// TIA Portal V15.1 export
// export: Created 2024-06-21T08:40:52.3398927Z, ExportSetting WithDefaults, DisplayName Totally Integrated Automation Portal, DisplayVersion V15.1 Update 5, DisplayName TIA Portal Openness, DisplayVersion V15.1 Update 5, DisplayName SINAMICS Startdrive Advanced, DisplayVersion V15.1, DisplayName G130, G150, S120, S150, SINAMICS MV, S210, DisplayVersion V15.1, DisplayName G110M, G120, G120C, G120D, G120P, DisplayVersion V15.1, DisplayName STEP 7 Professional, DisplayVersion V15.1 Update 5, DisplayName STEP 7 Safety, DisplayVersion V15.1, DisplayName WinCC Professional, DisplayVersion V15.1 Update 5, DisplayName SIMATIC Visualization Architect, DisplayVersion V15.1
FUNCTION "F209230ZS01Logic" : Void   // FC7031, F_FBD
TITLE = Safety Inputs ZMProc / Safety Logic 209230ZS01
{ S7_Optimized_Access := 'TRUE' }
VERSION : 0.1
// stored: AutoNumber false, IsIECCheckEnabled false, UDAEnableTagReadback false
   VAR_TEMP   // added for the SCL form of the ladder/FBD networks
      _w1 : Bool;
   END_VAR
BEGIN

REGION Network 1: **** 4.4 - Machine Status - Calculation **** Emergency Stop OK
   // Emergency Stop Ok When All Safety Inputs Are Ok
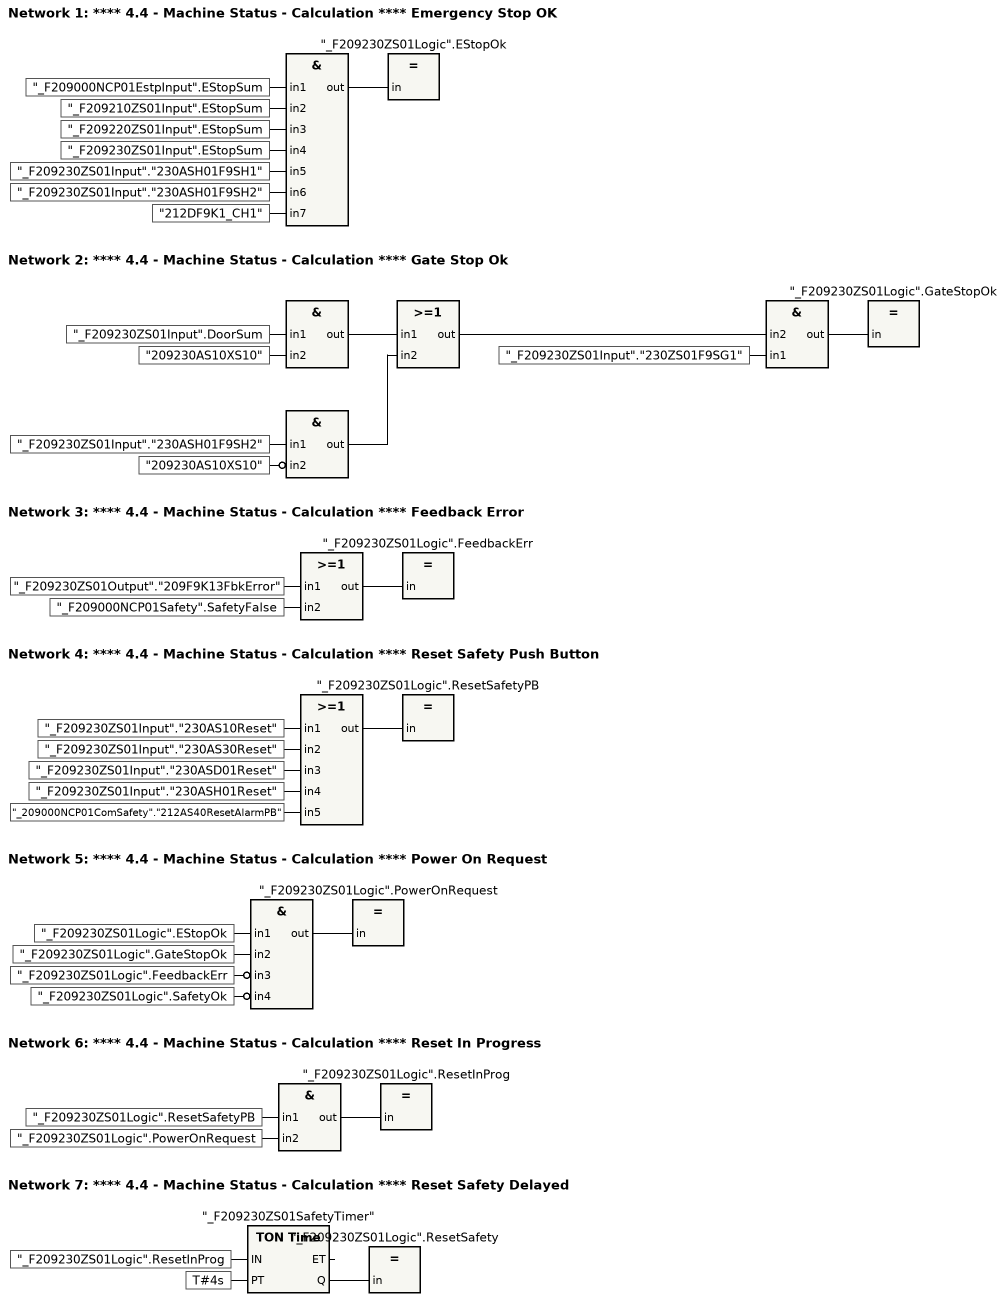
   "_F209230ZS01Logic".EStopOk := "_F209000NCP01EstpInput".EStopSum AND "_F209210ZS01Input".EStopSum AND "_F209220ZS01Input".EStopSum AND "_F209230ZS01Input".EStopSum AND "_F209230ZS01Input"."230ASH01F9SH1" AND "_F209230ZS01Input"."230ASH01F9SH2" AND "212DF9K1_CH1";
END_REGION

REGION Network 2: **** 4.4 - Machine Status - Calculation **** Gate Stop Ok
   // Gate Stop Ok
   "_F209230ZS01Logic".GateStopOk := (("_F209230ZS01Input".DoorSum AND "209230AS10XS10") OR ("_F209230ZS01Input"."230ASH01F9SH2" AND NOT "209230AS10XS10")) AND "_F209230ZS01Input"."230ZS01F9SG1";
END_REGION

REGION Network 3: **** 4.4 - Machine Status - Calculation **** Feedback Error
   // Feedback Error
   "_F209230ZS01Logic".FeedbackErr := "_F209230ZS01Output"."209F9K13FbkError" OR "_F209000NCP01Safety".SafetyFalse;
END_REGION

REGION Network 4: **** 4.4 - Machine Status - Calculation **** Reset Safety Push Button
   // Reset Safety Push Button
   "_F209230ZS01Logic".ResetSafetyPB := "_F209230ZS01Input"."230AS10Reset" OR "_F209230ZS01Input"."230AS30Reset" OR "_F209230ZS01Input"."230ASD01Reset" OR "_F209230ZS01Input"."230ASH01Reset" OR "_209000NCP01ComSafety"."212AS40ResetAlarmPB";
END_REGION

REGION Network 5: **** 4.4 - Machine Status - Calculation **** Power On Request
   // Power On Request
   "_F209230ZS01Logic".PowerOnRequest := "_F209230ZS01Logic".EStopOk AND "_F209230ZS01Logic".GateStopOk AND NOT "_F209230ZS01Logic".FeedbackErr AND NOT "_F209230ZS01Logic".SafetyOk;
END_REGION

REGION Network 6: **** 4.4 - Machine Status - Calculation **** Reset In Progress
   // Reset In Progress
   "_F209230ZS01Logic".ResetInProg := "_F209230ZS01Logic".ResetSafetyPB AND "_F209230ZS01Logic".PowerOnRequest;
END_REGION

REGION Network 7: **** 4.4 - Machine Status - Calculation **** Reset Safety Delayed
   // Reset Safety Delayed
   "_F209230ZS01SafetyTimer".TON(IN := "_F209230ZS01Logic".ResetInProg, PT := T#4s);
   "_F209230ZS01Logic".ResetSafety := "_F209230ZS01SafetyTimer".Q;
END_REGION

REGION Network 8: **** 4.4 - Machine Status - Calculation **** Power On
   // Power On
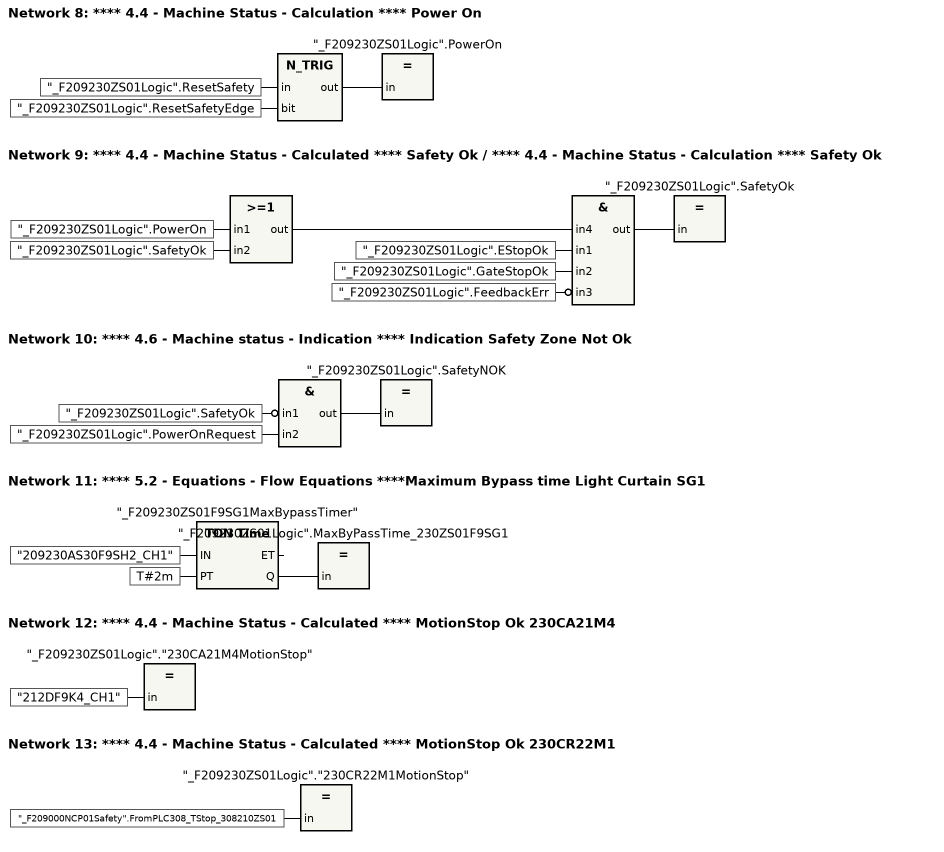
   #_w1 := NOT "_F209230ZS01Logic".ResetSafety AND "_F209230ZS01Logic".ResetSafetyEdge;   // falling edge
   "_F209230ZS01Logic".ResetSafetyEdge := "_F209230ZS01Logic".ResetSafety;
   "_F209230ZS01Logic".PowerOn := #_w1;
END_REGION

REGION Network 9: **** 4.4 - Machine Status - Calculated **** Safety Ok / **** 4.4 - Machine Status - Calculation **** Safety Ok
   // All safety is ok
   "_F209230ZS01Logic".SafetyOk := ("_F209230ZS01Logic".PowerOn OR "_F209230ZS01Logic".SafetyOk) AND "_F209230ZS01Logic".EStopOk AND "_F209230ZS01Logic".GateStopOk AND NOT "_F209230ZS01Logic".FeedbackErr;
END_REGION

REGION Network 10: **** 4.6 - Machine status - Indication **** Indication Safety Zone Not Ok
   // Indication Safety Zone Not Ok
   "_F209230ZS01Logic".SafetyNOK := NOT "_F209230ZS01Logic".SafetyOk AND "_F209230ZS01Logic".PowerOnRequest;
END_REGION

REGION Network 11: **** 5.2 - Equations - Flow Equations ****Maximum Bypass time Light Curtain SG1
   // Maximum Bypass time (Return Key Operation) for Light Curtain
   "_F209230ZS01F9SG1MaxBypassTimer".TON(IN := "209230AS30F9SH2_CH1", PT := T#2m);
   "_F209230ZS01Logic".MaxByPassTime_230ZS01F9SG1 := "_F209230ZS01F9SG1MaxBypassTimer".Q;
END_REGION

REGION Network 12: **** 4.4 - Machine Status - Calculated **** MotionStop Ok 230CA21M4
   // MotionStop Ok
   "_F209230ZS01Logic"."230CA21M4MotionStop" := "212DF9K4_CH1";
END_REGION

REGION Network 13: **** 4.4 - Machine Status - Calculated **** MotionStop Ok 230CR22M1
   // MotionStop Ok
   "_F209230ZS01Logic"."230CR22M1MotionStop" := "_F209000NCP01Safety".FromPLC308_TStop_308210ZS01;
END_REGION
END_FUNCTION
